// TwinCAT 3 PLC project Untitled1
// ProgramVersion: 3.1.4023.0
// libraries:
//   Tc2_Standard, * (Beckhoff Automation GmbH)
//   Tc2_System, * (Beckhoff Automation GmbH)
//   Tc3_Module, * (Beckhoff Automation GmbH)
// project tree:
//   GVLs/Blower/ Blower.TcGVL
//   GVLs/Counter/ CountUp.TcGVL
//   GVLs/LightBulb/ LightBulb.TcGVL
//   GVLs/PumpControl/ Pump.TcGVL
//   GVLs/Timers/ LEDTimer.TcGVL
//   / PlcTask.TcTTO
//   POUs/Application/ IO.TcPOU
//   POUs/Blower Controls/ Controls.TcPOU
//   POUs/DigitalTank/ TankControl.TcPOU
//   POUs/FunctionBlocks/ Blink.TcPOU
//   POUs/Lightbulb/ LightBulbCount.TcPOU, LightBulbTimer.TcPOU
//   POUs/ MAIN.TcPOU
//   POUs/Setup/ Alarm_Logic.TcPOU
//   VISUs/Image/ ImagePool.TcIPO (not stored)

CONFIGURATION Untitled1
    RESOURCE PLC ON TwinCAT3
        TASK PlcTask(INTERVAL := T#10ms, PRIORITY := 20);
        PROGRAM MAIN WITH PlcTask : MAIN;
    END_RESOURCE
END_CONFIGURATION

// ---- GVLs/Blower/Blower.TcGVL
{attribute 'qualified_only'}
VAR_GLOBAL
	
	// Inputs
	OnPushBTN		:	BOOL;
	OffPushBTN		:	BOOL;
	AutoPushBTN		:	BOOL;
	
	// Outputs
	AirBlowerPower	:	BOOL;
	BlowerStatus	:	ARRAY[1..2] OF BOOL;
	
END_VAR

// ---- GVLs/Counter/CountUp.TcGVL
{attribute 'qualified_only'}
VAR_GLOBAL
	Count	:	CTU;
END_VAR

// ---- GVLs/LightBulb/LightBulb.TcGVL
{attribute 'qualified_only'}
VAR_GLOBAL
	
	(* Input *)
	StartSwitch				:	BOOL;
	StopSwitch				:	BOOL;
	StartSignal				:	BOOL;
	StopSignal				:	BOOL;
	
	(* Output *)
	YellowLED		AT%Q*	:	BOOL	:= FALSE;
	
	
END_VAR

// ---- GVLs/PumpControl/Pump.TcGVL
{attribute 'qualified_only'}
VAR_GLOBAL

		HHSwitch	:	BOOL;
		HSwitch		:	BOOL;
		
		LLSwicth	:	BOOL;
		LSwitch		:	BOOL;
		
		Pump		:	BOOL;
		Valve		:	BOOL;
		
		YellowLED	:	BOOL;
		RedLED		:	BOOL;
		BlueLED		:	BOOL;
		
END_VAR

// ---- GVLs/Timers/LEDTimer.TcGVL
{attribute 'qualified_only'}
VAR_GLOBAL
	On_DelayLED		:	TON;
	Off_DelayLED	:	TOF;
END_VAR

// ---- POUs/MAIN.TcPOU
PROGRAM MAIN
VAR
END_VAR

LightBulbTimer();
Controls();
TankControl();
Alarm_Logic();

END_PROGRAM

// ---- POUs/Lightbulb/LightBulbTimer.TcPOU
PROGRAM LightBulbTimer
VAR
	ONS :	BOOL;
END_VAR

IO();
(*Delays the LED for 10 seconds to turn on *)
//LEDTimer.On_DelayLED  (IN	:=	LightBulb.StartSignal = TRUE,  PT	:=	T#10S, Q=> , ET => );
//LEDTimer.Off_DelayLED (IN	:=	LightBulb.StopSignal = TRUE, PT	:=	T#10S,	Q=>, ET=> );


IF Lightbulb.StartSignal AND ONS THEN
	
	Lightbulb.YellowLED		:=	TRUE;
	Lightbulb.StopSignal	:=	FALSE;
	
END_IF

IF Lightbulb.StopSignal AND ONS = FALSE THEN

	Lightbulb.YellowLED		:=	FALSE;	
	Lightbulb.StartSignal	:=	FALSE;

END_IF

END_PROGRAM

// ---- POUs/Application/IO.TcPOU
PROGRAM IO
VAR
END_VAR


LightBulb.StartSwitch 	:=	LightBulb.StartSignal;
LightBulb.StopSwitch	:=	LightBulb.StopSignal;

END_PROGRAM

// ---- POUs/Blower Controls/Controls.TcPOU
PROGRAM Controls
VAR
	MainState	:	INT;// 0 : OFF || 1 : manual Mode | 2 : AutoMode
END_VAR


IF Blower.OnPushBTN AND Blower.AutoPushBTN = FALSE AND Blower.AutoPushBTN = FALSE AND MainState <> 2 THEN
	
	MainState				:=	1;
	
END_IF

IF Blower.OffPushBTN THEN
	
	Mainstate				:=	0;
	Blower.AirBlowerPower	:=	FALSE;
	Blower.AutoPushBTN		:=	FALSE;
	Blower.OnPushBTN		:=	FALSE;
	
END_IF

IF Blower.AutoPushBTN AND Blower.OffPushBTN = FALSE AND Blower.OnPushBTN = FALSE THEN
	
	MainState 				:=	2;
	
END_IF

IF (Blower.OnPushBTN OR Blower.AutoPushBTN) AND Blower.OffPushBTN = FALSE  THEN
	
	Blower.AirBlowerPower	:=	TRUE;
	
END_IF

END_PROGRAM

// ---- POUs/DigitalTank/TankControl.TcPOU
PROGRAM TankControl
VAR
	MainState	:	INT;
	FillModeDelay		:	TON;
	DrainModeDelay		:	TON;
END_VAR

FillModeDelay(IN := Pump.LSwitch, PT := T#10S, Q=>,ET=>);
DrainModeDelay(IN := Pump.HSwitch, PT := T#10S, Q=>,ET=>);

IF Pump.LSwitch AND Pump.HSwitch = FALSE THEN
	
	Pump.Pump	:=	FillModeDelay.Q;
	Pump.Valve	:=	FALSE;
	
END_IF

IF Pump.HSwitch AND Pump.LSwitch = FALSE THEN
	
	Pump.Pump	:=	FALSE;
	Pump.Valve	:=	DrainModeDelay.Q;
	
END_IF

END_PROGRAM

// ---- POUs/Setup/Alarm_Logic.TcPOU
PROGRAM Alarm_Logic
VAR
	
	RedStack		:	Blink;
	YellowStack		:	Blink;
	BlueStack		:	Blink;
	YellowLED		:	Blink;
	
END_VAR


IF Pump.LLSwicth AND Pump.HHSwitch = FALSE THEN

	RedStack(Enable := TRUE, Period := T#125MS ,Q=> Pump.RedLED);
	YellowStack(Enable := TRUE, Period := T#125MS ,Q=> Pump.YellowLED);	

END_IF

END_PROGRAM

// ---- POUs/FunctionBlocks/Blink.TcPOU
FUNCTION_BLOCK Blink
VAR_INPUT

	Enable		:	BOOL;	(* Enable Bit to Start Running *)

	Period		:	TIME;	(* Period for Flashing *)

END_VAR


(* === Output Variables === *)
VAR_OUTPUT

	Q		:	BOOL;	(* Flasher Output Bit *)

END_VAR


(* === Local Variables === *)
VAR

	onPeriod	:	Ton;	(* on Period Timer *)

	offPeriod	:	Ton;	(* off Period Timer *)

END_VAR

VAR ConSTANT
END_VAR



IF Enable = TRUE THEN
	
	OnPeriod(IN := NOT OffPeriod.Q, PT := Period/2);
	OnPeriod(IN := OnPeriod.Q, PT := Period/2);
	
	Q	:=	NOT OnPeriod.Q;
	
END_IF

END_FUNCTION_BLOCK

// ---- POUs/Lightbulb/LightBulbCount.TcPOU
PROGRAM LightBulbCount
VAR
	ResetBTN: BOOL;
END_VAR

(*Counter TURN ON 5 times until LED can actually turn on*)

(*CountUp.Count (CU := LightBulb.LightSwitch, RESET := ResetBTN, PV := 5, Q=>, CV=> );

IF LightBulb.LightSwitch THEN
	LightBulb.YellowLED	:=	CountUp.Count.Q;
END_IF

*)

END_PROGRAM
